{attribute 'qualified_only'}
// Robot6 --joints parameters of setup arms
VAR_GLOBAL
	// absolute encoder value at minimal joint positon
	g_minLinkEncoder :ARRAY[1..g_cartJntNum] OF DINT :=[0, 0, 0, 0, 12912698, 863216, 13187303, 654894];
		 
	// absolute encoder value at maximum joint positon
	g_maxLinkEncoder :ARRAY[1..g_cartJntNum] OF DINT :=[0, 0, 0, 0, 10127418, 3841586, 15255509,16569304 ];
	
	// absolute encoder value at calibrated positon
	g_caliLinkEncoder :ARRAY[1..g_cartJntNum] OF DINT :=[0, 0, 0, 0, 12912698, 2352401, 15255509, 8612099];
	
	 // if absolute encoder value cross zeros within joint motion range
	g_linkEncZeroCross :ARRAY[1..g_cartJntNum] OF INT :=[0, 0, 0, 0, 0, 0, 0, 1];
		 

	// abolute encoder expanded limit buffer in case there is calibrtion error at limit position
	g_linkEncLimitBuffer : DINT := 100000;

	// absolute encoder direction
	g_asbEncoderDir :ARRAY[1..g_cartJntNum] OF INT :=[1, 1, 1, 1, -1, 1, -1, -1];
													
	// flag if joint can rotate multiple cycles
	g_multipleCyclesJoint :ARRAY[1..g_cartJntNum] OF INT :=[0, 0, 0, 0, 0, 0, 0, 0];
		 
	// joint position at link encoder calibrated point
	g_linkEncCaliJntPos :ARRAY[1..g_cartJntNum] OF LREAL :=[0.0, 0.0, 0.0, 0.0, 0.0, 0.0, 0, 0.0];
	
	 // joint SDO address
	g_slaveCartNetID: T_AmsNetId:='169.254.186.39.7.1';
	g_slaveCartJointNetPort:ARRAY[1..g_cartJntNum] OF UINT :=[1005,	1004,	1003,	1002,	1001,   1006,  1007,  1008];

END_VAR

(* stored: Version 1.1.0.1, ProductVersion 3.1.4024.11
   GVL GVL_CartJointEncoderCaliData_6: Id {57256aba-e142-41c1-94fd-1676368502f4} *)
